(* IEC 61131-3 sources: DatObjWrap/src/Ar/DatObjWrap, 6 files *)

(* ---- DatObjWrap.typ ---- *)
(*
 * File: DatObjWrap.typ
 * Copyright (c) 2023 Loupe
 * https://loupe.team
 *
 * This file is part of DatObjWrap, licensed under the MIT License.
 *
  ********************************************************************
 * Data types of library DatObjWrap
 ********************************************************************)

TYPE
	DOWRAP_OP_enum :
		(
		DOWRAP_OP_INVALID := 0,
		DOWRAP_OP_OPEN,
		DOWRAP_OP_SAVEAS
		);
	DOWRAP_ST_enum :
		(
		DOWRAP_ST_WAIT := 0, (*0*)
		DOWRAP_ST_GETINFO, (*1*)
		DOWRAP_ST_CREATE, (*2*)
		DOWRAP_ST_OPEN, (*3*)
		DOWRAP_ST_SAVE, (*4*)
		DOWRAP_ST_ERROR := 999, (*999*)
		DOWRAP_ST_
		);
	DatObjWrap_Int_FUB_typ : 	STRUCT
		DatObjGetInfo : DatObjInfo;
		DatObjCreate : DatObjCreate;
		DatObjWrite : DatObjWrite;
		DatObjRead : DatObjRead;
	END_STRUCT;
	DatObjWrap_Internal_typ : 	STRUCT
		Ident : UDINT; (*Data object ident*)
		State : DINT; (*State variable*)
		CurrOperation : DINT; (*Current operation (Save or Load)*)
		FUB : DatObjWrap_Int_FUB_typ;
		CMD : DatObjWrap_IN_CMD_typ;
	END_STRUCT;
	DatObjWrap_OUT_STAT_typ : 	STRUCT
		Busy : BOOL; (*Object is busy performing an action*)
		Done : BOOL; (*Action finished successfully*)
		Error : BOOL; (*There is an error with the DOHandling*)
		ErrorID : UINT; (*Error number from internal FUBs*)
		ErrorString : STRING[DOWRAP_STRLEN_ERROR];
		ErrorLevel : USINT;
		ErrorState : DINT; (*State in which error occurred*)
	END_STRUCT;
	DatObjWrap_OUT_typ : 	STRUCT
		STAT : DatObjWrap_OUT_STAT_typ;
	END_STRUCT;
	DatObjWrap_IN_PAR_typ : 	STRUCT
		DataObjName : STRING[8]; (*Name of the data object to which to store data*)
		pData : UDINT; (*Pointer to the data location to be saved from/loaded to*)
		len : UDINT; (*Length of the data to be saved/loaded*)
	END_STRUCT;
	DatObjWrap_IN_CMD_typ : 	STRUCT
		Open : BOOL; (*Load settings from Data Object.*)
		SaveAs : BOOL; (*Save settings to Data Object.*)
		AcknowledgeError : BOOL; (*Acknowledge errors*)
	END_STRUCT;
	DatObjWrap_IN_typ : 	STRUCT
		CMD : DatObjWrap_IN_CMD_typ;
		PAR : DatObjWrap_IN_PAR_typ;
	END_STRUCT;
	DatObjWrap_typ : 	STRUCT
		IN : DatObjWrap_IN_typ;
		OUT : DatObjWrap_OUT_typ;
		Internal : DatObjWrap_Internal_typ;
	END_STRUCT;
END_TYPE

(* ---- DatObjWrap.fun ---- *)
(*
 * File: DatObjWrap.fun
 * Copyright (c) 2023 Loupe
 * https://loupe.team
 *
 * This file is part of DatObjWrap, licensed under the MIT License.
 *
  ********************************************************************
 * Functions and function blocks of library DatObjWrap
 ********************************************************************)

FUNCTION DatObjWrapFn_Cyclic : BOOL (*This function implements a wrapper for Data Object writing and reading.*)
	VAR_IN_OUT
		t : DatObjWrap_typ; (*Data object wrapper control object.*)
	END_VAR
END_FUNCTION

FUNCTION DatObjWrapOpen_Init : BOOL (*Synchronously loads a data object. Should ONLY be called in the INIT routine.*)
	VAR_IN_OUT
		t : DatObjWrap_typ; (*Data object wrapper control object.*)
	END_VAR
END_FUNCTION

FUNCTION dowSetError : BOOL (*Set error status on DatObjWrap*)
	VAR_INPUT
		ErrorID : UINT;
	END_VAR
	VAR_IN_OUT
		t : DatObjWrap_typ;
	END_VAR
END_FUNCTION

(* ---- DatObjWrapFn_Cyclic.st ---- *)
(*
 * File: DatObjWrapFn_Cyclic.st
 * Copyright (c) 2023 Loupe
 * https://loupe.team
 *
 * This file is part of DatObjWrap, licensed under the MIT License.
 *
  ********************************************************************
 * Implementation of library DatObjWrap
 ********************************************************************)

(****************************************************************************)
(* This function implements a wrapper for Data Object writing and reading	*)
(****************************************************************************)

(* Resetting internal CMDs				DONE and TESTED DFB 20110516 *)

(* Main state machine					DONE and TESTED DFB 20110516 *)

	(* ST_WAIT							DONE and TESTED DFB 20110516 *)
		(* Handling CMDs				DONE and TESTED DFB 20110516 *)
			(* Setting CurrOperation	DONE and TESTED DFB 20110516 *)
		(* Handling Done				DONE and TESTED DFB 20110516 *)

	(* ST_GETINFO						DONE and TESTED DFB 20110516 *)
		(* Handling FUB					DONE and TESTED DFB 20110516 *)
		(* Checking status				DONE and TESTED DFB 20110516 *)
			(* Done						DONE and TESTED DFB 20110516 *)
			(* No error					DONE and TESTED DFB 20110516 *)
			(* Module Not Found			DONE and TESTED DFB 20111222 *)
				(* Open					DONE and TESTED DFB 20111222 *)
				(* SaveAs				DONE and TESTED DFB 20110516 *)
			(* Other error				DONE will not be tested *)

	(* ST_CREATE						DONE and TESTED DFB 20110516 *)
		(* Handling FUB					DONE and TESTED DFB 20110516 *)
		(* Checking status				DONE and TESTED DFB 20110516 *)
			(* Done						DONE and TESTED DFB 20110516 *)
			(* No error					DONE and TESTED DFB 20110516 *)
			(* Other error				DONE and TESTED DFB 20111222 *)

	(* ST_OPEN							DONE and TESTED DFB 20110516 *)
		(* Handling FUB					DONE and TESTED DFB 20110516 *)
		(* Checking status				DONE and TESTED DFB 20110516 *)
			(* Done						DONE and TESTED DFB 20110516 *)
			(* No error					DONE and TESTED DFB 20110516 *)
			(* Other error				DONE and TESTED DFB 20111222 *)

	(* ST_SAVE							DONE and TESTED DFB 20110516 *)
		(* Handling FUB					DONE and TESTED DFB 20110516 *)
		(* Checking status				DONE and TESTED DFB 20110516 *)
			(* Done						DONE and TESTED DFB 20110516 *)
			(* No error					DONE and TESTED DFB 20110516 *)
			(* Other error				DONE and TESTED DFB 20111222 *)

	(* ST_ERROR							DONE and TESTED DFB 20111222 *)

(* Busy, Done, Error					DONE and TESTED DFB 20111222 *)

(* Resetting AcknowledgeError			DONE and TESTED DFB 20110516 *)

FUNCTION DatObjWrapFn_Cyclic

(****************************************************)
(* Set return value to get rid of compile warning 	*)
(****************************************************)

DatObjWrapFn_Cyclic:=	FALSE;

(****************************************************)
(* Reset Internal CMDs								*)
(****************************************************)

IF( NOT(t.IN.CMD.Open) )THEN

	t.Internal.CMD.Open:=	0;

END_IF

IF( NOT(t.IN.CMD.SaveAs) )THEN

	t.Internal.CMD.SaveAs:=	0;

END_IF

(****************************************)
(* Main State machine					*)
(****************************************)

CASE t.Internal.State OF

	DOWRAP_ST_WAIT:

		(* If all CMDs are cleared, then clear Done status *)

		IF( 	NOT(t.IN.CMD.Open)
			AND NOT(t.IN.CMD.SaveAs)
			)THEN

			t.OUT.STAT.Done:=	0;

		END_IF

		(* Set CurrOperation to INVALID. It will be set below on leaving the state *)

		t.Internal.CurrOperation:=	DOWRAP_OP_INVALID;

		(* Wait for new commands *)

		IF( t.IN.CMD.SaveAs AND NOT(t.Internal.CMD.SaveAs) )THEN

			t.Internal.CMD.SaveAs:=	1;

			t.OUT.STAT.Busy:=	1;
			t.OUT.STAT.Done:=	0;

			t.Internal.State:=			DOWRAP_ST_GETINFO;
			t.Internal.CurrOperation:=	DOWRAP_OP_SAVEAS;

		ELSIF( t.IN.CMD.Open AND NOT(t.Internal.CMD.Open) )THEN

			t.Internal.CMD.Open:=	1;

			t.OUT.STAT.Busy:=	1;
			t.OUT.STAT.Done:=	0;

			t.Internal.State:=			DOWRAP_ST_GETINFO;
			t.Internal.CurrOperation:=	DOWRAP_OP_OPEN;

		END_IF

	DOWRAP_ST_GETINFO:

		(* DatObjGetInfo *)

		t.Internal.FUB.DatObjGetInfo.enable:=	1;
		t.Internal.FUB.DatObjGetInfo.pName:=	ADR(t.IN.PAR.DataObjName);

		(* Check FUB status *)

		(* If finished *)

		IF( t.Internal.FUB.DatObjGetInfo.status < DOWRAP_STATUS_FUB_DISABLED ) THEN

			t.Internal.FUB.DatObjGetInfo.enable:=	0;

			(* if no error *)

			IF( t.Internal.FUB.DatObjGetInfo.status = 0 ) THEN

				(* store ident *)

				t.Internal.Ident:=	t.Internal.FUB.DatObjGetInfo.ident;

				(* go to appropriate state *)

				IF( t.Internal.CurrOperation = DOWRAP_OP_OPEN ) THEN

					t.Internal.State:=	DOWRAP_ST_OPEN;

				ELSIF( t.Internal.CurrOperation = DOWRAP_OP_SAVEAS ) THEN

					t.Internal.State:=	DOWRAP_ST_SAVE;

				ELSE

					t.Internal.State:=	DOWRAP_ST_WAIT;

				END_IF

			(* if data object not found *)

			ELSIF( t.Internal.FUB.DatObjGetInfo.status = doERR_MODULNOTFOUND )THEN

				(* if loading, then an error *)

				IF( t.Internal.CurrOperation = DOWRAP_OP_OPEN ) THEN

					dowSetError( t.Internal.FUB.DatObjGetInfo.status, t );

				ELSIF( t.Internal.CurrOperation = DOWRAP_OP_SAVEAS ) THEN

					t.Internal.State:=	DOWRAP_ST_CREATE;

				ELSE

					t.Internal.State:=	DOWRAP_ST_WAIT;

				END_IF

			(* if other error *)

			ELSE

				dowSetError( t.Internal.FUB.DatObjGetInfo.status, t );

			END_IF(* status checking *)

		END_IF(* if FUB finished *)

	DOWRAP_ST_CREATE:

		(* Create the data object and write to it *)
		(* Will only get here if saving *)

		t.Internal.FUB.DatObjCreate.enable:=	1;
		t.Internal.FUB.DatObjCreate.grp:=		0;
		t.Internal.FUB.DatObjCreate.pName:=		ADR(t.IN.PAR.DataObjName);
		t.Internal.FUB.DatObjCreate.len:=		t.IN.PAR.len;
		t.Internal.FUB.DatObjCreate.MemType:=	doUSRROM;
		t.Internal.FUB.DatObjCreate.Option:=	0;
		t.Internal.FUB.DatObjCreate.pCpyData:=	t.IN.PAR.pData;

		(* Check FUB status *)

		(* if FUB finished *)

		IF( t.Internal.FUB.DatObjCreate.status < DOWRAP_STATUS_FUB_DISABLED ) THEN

			t.Internal.FUB.DatObjCreate.enable:=	0;

			(* if no error *)

			IF( t.Internal.FUB.DatObjCreate.status = 0 ) THEN

				(* Done saving *)

				t.OUT.STAT.Busy:=	0;
				t.OUT.STAT.Done:=	1;

				t.Internal.State:=	DOWRAP_ST_WAIT;

			(* if other error *)

			ELSE

				dowSetError( t.Internal.FUB.DatObjCreate.status, t );

//				t.OUT.STAT.Error:=		1;
//				t.OUT.STAT.ErrorID:=	t.Internal.FUB.DatObjCreate.status;
//				t.OUT.STAT.ErrorState:=	t.Internal.State;
//				t.Internal.State:=		DOWRAP_ST_ERROR;

			END_IF(* status checking *)

		END_IF(* if FUB finished *)

	DOWRAP_ST_OPEN:

		(* Read data from data object *)

		t.Internal.FUB.DatObjRead.enable:=			1;
		t.Internal.FUB.DatObjRead.ident:=			t.Internal.Ident;
		t.Internal.FUB.DatObjRead.Offset:=			0;
		t.Internal.FUB.DatObjRead.pDestination:=	t.IN.PAR.pData;
		t.Internal.FUB.DatObjRead.len:=				t.IN.PAR.len;

		(* Check FUB status *)

		(* If finished *)

		IF( t.Internal.FUB.DatObjRead.status < DOWRAP_STATUS_FUB_DISABLED ) THEN

  			t.Internal.FUB.DatObjRead.enable:=	0;

  			(* if no error *)

			IF( t.Internal.FUB.DatObjRead.status = 0 ) THEN

				(* Done loading *)

				t.OUT.STAT.Busy:=	0;
				t.OUT.STAT.Done:=	1;

				t.Internal.State:=	DOWRAP_ST_WAIT;

			(* if other error *)

			ELSE

				dowSetError( t.Internal.FUB.DatObjRead.status, t );

//				t.OUT.STAT.Error:=		1;
//				t.OUT.STAT.ErrorID:=	t.Internal.FUB.DatObjRead.status;
//				t.OUT.STAT.ErrorState:=	t.Internal.State;
//				t.Internal.State:=		DOWRAP_ST_ERROR;

			END_IF(* status checking *)

		END_IF(* if FUB finished *)

	DOWRAP_ST_SAVE:

		(* Write data to data object *)

		t.Internal.FUB.DatObjWrite.enable:=		1;
		t.Internal.FUB.DatObjWrite.ident:=		t.Internal.Ident;
		t.Internal.FUB.DatObjWrite.Offset:=		0;
		t.Internal.FUB.DatObjWrite.pSource:=	t.IN.PAR.pData;
		t.Internal.FUB.DatObjWrite.len:=		t.IN.PAR.len;

		(* Check FUB status *)

		(* if finished *)

		IF( t.Internal.FUB.DatObjWrite.status < DOWRAP_STATUS_FUB_DISABLED ) THEN

			t.Internal.FUB.DatObjWrite.enable:=	0;

  			(* if no error *)

			IF( t.Internal.FUB.DatObjWrite.status = 0 ) THEN

				(* Done saving *)

				t.OUT.STAT.Busy:=	0;
				t.OUT.STAT.Done:=	1;

				t.Internal.State:=	DOWRAP_ST_WAIT;

			(* if other error *)

			ELSE

				dowSetError( t.Internal.FUB.DatObjWrite.status, t );

//				t.OUT.STAT.Error:=		1;
//				t.OUT.STAT.ErrorID:=	t.Internal.FUB.DatObjWrite.status;
//				t.OUT.STAT.ErrorState:=	t.Internal.State;
//				t.Internal.State:=		DOWRAP_ST_ERROR;

			END_IF(* status checking *)

		END_IF(* if FUB finished *)

	DOWRAP_ST_ERROR:

		IF( t.IN.CMD.AcknowledgeError )THEN

			t.IN.CMD.AcknowledgeError:=	0;

			t.OUT.STAT.Error:=			0;
			t.OUT.STAT.ErrorID:=		0;
			t.OUT.STAT.ErrorString:=	'';
			t.OUT.STAT.ErrorLevel:=		0;
			t.OUT.STAT.ErrorState:=		0;

			t.Internal.State:=		DOWRAP_ST_WAIT;

		END_IF

END_CASE

(* Reset AcknowledgeError CMD *)

t.IN.CMD.AcknowledgeError:=	0;

(****************************************)
(* Call FUBs							*)
(****************************************)

t.Internal.FUB.DatObjGetInfo();
t.Internal.FUB.DatObjCreate();
t.Internal.FUB.DatObjRead();
t.Internal.FUB.DatObjWrite();

END_FUNCTION

(* ---- DatObjWrapOpen_Init.st ---- *)
(*
 * File: DatObjWrapOpen_Init.st
 * Copyright (c) 2023 Loupe
 * https://loupe.team
 *
 * This file is part of DatObjWrap, licensed under the MIT License.
 *
  ********************************************************************
 * Implementation of library DatObjWrap
 ********************************************************************)

(************************************************************************************)
(* Synchronously loads a data object. Should ONLY be called in the INIT routine.	*)
(************************************************************************************)

(* GetInfo			DONE and TESTED DFB 20110516 *)
	(* No error		DONE and TESTED DFB 20110516 *)
	(* Error		DONE and TESTED DFB 20111222 *)

(* Read				DONE and TESTED DFB 20110516 *)
	(* No error		DONE and TESTED DFB 20110516 *)
	(* Error		DONE and TESTED DFB 20111222 *)

FUNCTION DatObjWrapOpen_Init

(****************************************************)
(* Set return value to get rid of compile warning 	*)
(****************************************************)

DatObjWrapOpen_Init:=	FALSE;

(********************************************)
(* DatObjGetInfo 							*)
(********************************************)

(* Map inputs *)

t.Internal.FUB.DatObjGetInfo.enable:=	1;
t.Internal.FUB.DatObjGetInfo.pName:=	ADR(t.IN.PAR.DataObjName);

(* Call FUB *)

t.Internal.FUB.DatObjGetInfo();

t.Internal.FUB.DatObjGetInfo.enable:=	0;

(* check status *)

(* if no error *)

IF( t.Internal.FUB.DatObjGetInfo.status = 0 ) THEN

	(* store ident *)

	t.Internal.Ident:=	t.Internal.FUB.DatObjGetInfo.ident;

(* Error *)

ELSE

	(* Set error info and return *)

	dowSetError( t.Internal.FUB.DatObjGetInfo.status, t );

	RETURN;

END_IF

(********************************************)
(* DatObjRead	 							*)
(********************************************)

(* Map inputs *)

t.Internal.FUB.DatObjRead.enable:=			1;
t.Internal.FUB.DatObjRead.ident:=			t.Internal.Ident;
t.Internal.FUB.DatObjRead.Offset:=			0;
t.Internal.FUB.DatObjRead.pDestination:=	t.IN.PAR.pData;
t.Internal.FUB.DatObjRead.len:=				t.IN.PAR.len;

(* Call FUB *)

t.Internal.FUB.DatObjRead();

t.Internal.FUB.DatObjRead.enable:=	0;

(* check status *)

(* If Error *)

IF( t.Internal.FUB.DatObjRead.status <> 0 ) THEN

	(* Set error info and return *)

	dowSetError( t.Internal.FUB.DatObjRead.status, t );

	RETURN;

END_IF

END_FUNCTION

(* ---- dowSetError.st ---- *)
(*
 * File: dowSetError.st
 * Copyright (c) 2023 Loupe
 * https://loupe.team
 *
 * This file is part of DatObjWrap, licensed under the MIT License.
 *
  ********************************************************************
 * Implementation of library DatObjWrap
 ********************************************************************)

(********************************************************************)
(* Set error status on DatObjWrap 									*)
(********************************************************************)

(* Reset Busy, Done			DONE and TESTED DFB 20111222 *)
(* Set Error				DONE and TESTED DFB 20111222 *)
(* Set ErrorID				DONE and TESTED DFB 20111222 *)
(* Set ErrorLevel			DONE and TESTED DFB 20111222 *)
(* Set ErrorState			DONE and TESTED DFB 20111222 *)
(* Set State				DONE and TESTED DFB 20111222 *)
(* Set ErrorString			DONE and TESTED DFB 20111222 *)

FUNCTION dowSetError

(****************************************************)
(* Set return value to get rid of compile warning 	*)
(****************************************************)

dowSetError:=	FALSE;

(************************************************)
(* Set error status								*)
(************************************************)

t.OUT.STAT.Busy:=		0;
t.OUT.STAT.Done:=		0;
t.OUT.STAT.Error:=		1;
t.OUT.STAT.ErrorID:=	ErrorID;
t.OUT.STAT.ErrorLevel:=	3;
t.OUT.STAT.ErrorState:=	t.Internal.State;
t.Internal.State:=		DOWRAP_ST_ERROR;

(* Set ErrorString *)

CASE ErrorID OF

	0: t.OUT.STAT.ErrorString:=	'';

	doERR_ILLPARAMETER:			t.OUT.STAT.ErrorString:=	'Invalid parameter. Check IN.PAR.pData.';
	doERR_DUPOBJECT:			t.OUT.STAT.ErrorString:=	'Object already present.';
	doERR_ILLMEMTYPE:			t.OUT.STAT.ErrorString:=	'Invalid memory type.';
	doERR_NOMEMORY:				t.OUT.STAT.ErrorString:=	'No memory available for object.';
	doERR_BRINSTALL:			t.OUT.STAT.ErrorString:=	'Error installing data object.';
	doERR_ILLOBJECT:			t.OUT.STAT.ErrorString:=	'Data object not found. Check IN.PAR.DataObjName.';
	doERR_ILLOBJTYPE:			t.OUT.STAT.ErrorString:=	'Object found, but it was not a data object. Check IN.PAR.DataObjName.';
	doERR_WRONGOFFSET:			t.OUT.STAT.ErrorString:=	'Invalid offset specified.';
	doERR_ILLEGALLENGTH:		t.OUT.STAT.ErrorString:=	'Invalid length specified. Check IN.PAR.len.';
	doERR_MODULNOTFOUND:		t.OUT.STAT.ErrorString:=	'Data object not found. Check IN.PAR.DataObjName.';
	doERR_WRONGTIME:			t.OUT.STAT.ErrorString:=	'Invalid date set.';
	doERR_ILLSTATE:				t.OUT.STAT.ErrorString:=	'Data object not in correct state.';
	doERR_STARTHANDLER:			t.OUT.STAT.ErrorString:=	'System error.';
	doERR_TOOLONG_MODULNAME:	t.OUT.STAT.ErrorString:=	'Data object name is too long. Check IN.PAR.DataObjName.';
	doERR_BURNINGOBJECT:		t.OUT.STAT.ErrorString:=	'System error.';

	ELSE	t.OUT.STAT.ErrorString:=	'Unknown error.';

END_CASE

END_FUNCTION

(* ---- DatObjWrap.var ---- *)
(*
 * File: DatObjWrap.var
 * Copyright (c) 2023 Loupe
 * https://loupe.team
 *
 * This file is part of DatObjWrap, licensed under the MIT License.
 *
  ********************************************************************
 * Constants of library DatObjWrap
 ********************************************************************)
VAR CONSTANT
	DOWRAP_STATUS_FUB_DISABLED : UINT := 65534;
	DOWRAP_STRLEN_ERROR : USINT := 80;
END_VAR
